# EPICS autosave request: iocBoot/auto_settings.req
$(P)AO:1-SP
$(P)AO:2-SP
$(P)AO:3-SP
$(P)AO:4-SP
$(P)AO:5-SP
$(P)AO:6-SP
$(P)AO:7-SP
$(P)AO:8-SP
